(* IEC 61131-3 sources: rules_plc/examples/st_c_implementation, 3 files *)

(* ---- base.st ---- *)
FUNCTION_BLOCK BASE_FB
    VAR_INPUT
        xTrigger: BOOL;
    END_VAR
    VAR_OUTPUT
        xDone: BOOL;
    END_VAR

    xDone := xTrigger;

END_FUNCTION_BLOCK

(* ---- mid.st ---- *)
(* {external} FUNCTION_BLOCK declared here; the body is provided by
mid.cc as a native C++ definition. plc emits only an extern
declaration for EXT_FB and skips code generation for its body. *)

{external}
FUNCTION_BLOCK EXT_FB
    VAR_INPUT
        rIn: REAL;
    END_VAR
    VAR_OUTPUT
        rOut: REAL;
    END_VAR
    VAR
        base: BASE_FB;
    END_VAR
END_FUNCTION_BLOCK

(* ---- main_program.st ---- *)
PROGRAM main_program
    VAR
        fbBase: BASE_FB;
        fbExt:  EXT_FB;
    END_VAR

    fbBase(xTrigger := TRUE);
    fbExt(rIn := 1.0);

END_PROGRAM
